(* IEC 61131-3 sources: eCockpitGit/test_project/src/%F%03 Module/%POU%FB_Module/%F%SYS Values/%PRO%SYS_valueAccess, 1 file *)

(* ---- %GETSET%Get.st ---- *)
VAR
END_VAR

(*%!%__DELIMITER__%!%*)
SYS_valueAccess		:=		EValueAccess.none;
